FUNCTION_BLOCK Control (* Composite Function Block Type *)
  (* Standard: 61499-2 *)
  (* Version 0.0, 6/3/2016, Andrei, nxtControl GmbH, template *)
  PACKAGE Main;
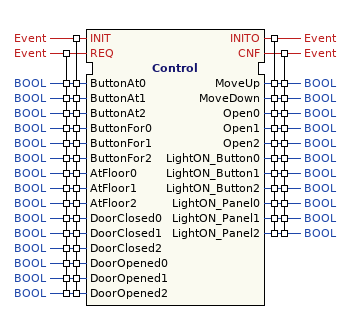
  EVENT_INPUT
    INIT WITH ButtonAt0, ButtonAt1, ButtonAt2, ButtonFor0, ButtonFor1, ButtonFor2, AtFloor0, AtFloor1, AtFloor2, DoorClosed0, DoorClosed1, DoorClosed2, DoorOpened0, DoorOpened1, DoorOpened2; (* Initialization Request *)
    REQ WITH ButtonAt0, ButtonAt1, ButtonAt2, ButtonFor0, ButtonFor1, ButtonFor2, AtFloor0, AtFloor1, AtFloor2, DoorClosed0, DoorClosed1, DoorClosed2, DoorOpened0, DoorOpened1, DoorOpened2; (* Normal Execution Request *)
  END_EVENT
  EVENT_OUTPUT
    INITO WITH MoveUp, MoveDown, Open0, Open1, Open2, LightON_Button0, LightON_Button1, LightON_Button2, LightON_Panel0, LightON_Panel1, LightON_Panel2; (* Initialization Confirm *)
    CNF WITH MoveUp, MoveDown, Open0, Open1, Open2, LightON_Button0, LightON_Button1, LightON_Button2, LightON_Panel0, LightON_Panel1, LightON_Panel2; (* Execution Confirmation *)
  END_EVENT
  VAR_INPUT
    ButtonAt0 : BOOL;
    ButtonAt1 : BOOL;
    ButtonAt2 : BOOL;
    ButtonFor0 : BOOL;
    ButtonFor1 : BOOL;
    ButtonFor2 : BOOL;
    AtFloor0 : BOOL; (* Input event qualifier *)
    AtFloor1 : BOOL;
    AtFloor2 : BOOL;
    DoorClosed0 : BOOL;
    DoorClosed1 : BOOL;
    DoorClosed2 : BOOL;
    DoorOpened0 : BOOL;
    DoorOpened1 : BOOL;
    DoorOpened2 : BOOL;
  END_VAR
  VAR_OUTPUT
    MoveUp : BOOL; (* Output event qualifier *)
    MoveDown : BOOL;
    Open0 : BOOL;
    Open1 : BOOL;
    Open2 : BOOL;
    LightON_Button0 : BOOL;
    LightON_Button1 : BOOL;
    LightON_Button2 : BOOL;
    LightON_Panel0 : BOOL;
    LightON_Panel1 : BOOL;
    LightON_Panel2 : BOOL;
  END_VAR
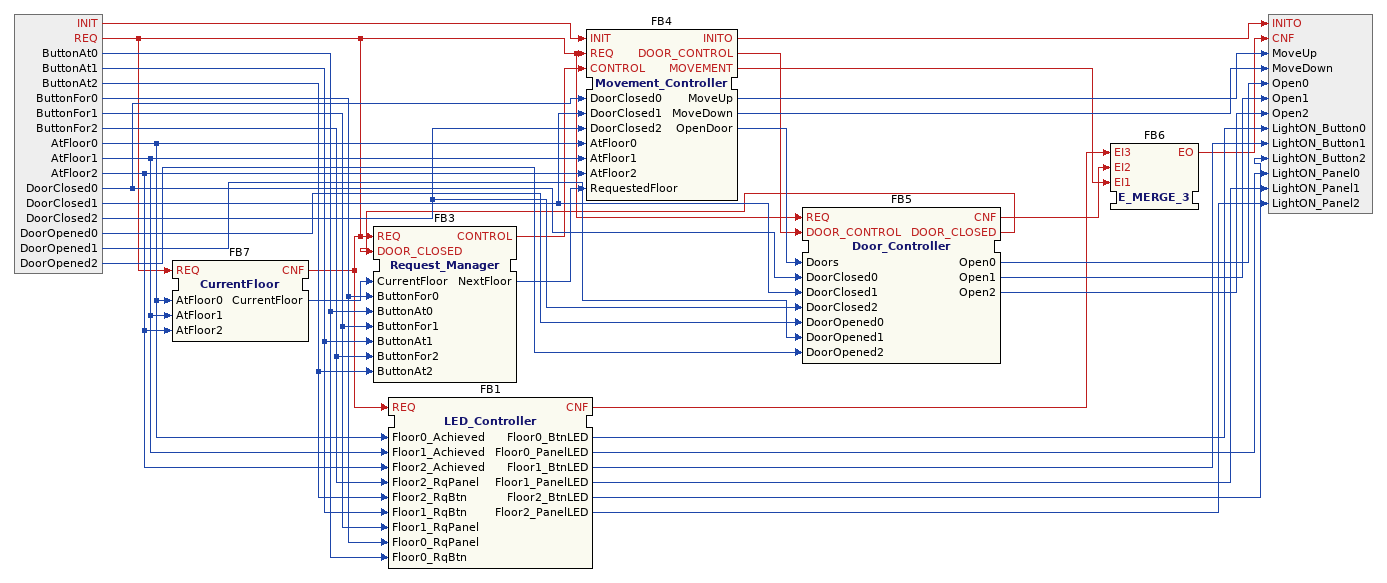
  FBS
    FB1 : LED_Controller;
    FB4 : Movement_Controller;
    FB5 : Door_Controller;
    FB6 : E_MERGE_3;
    FB3 : Request_Manager;
    FB7 : CurrentFloor;
  END_FBS
  EVENT_CONNECTIONS
    REQ TO FB1.REQ;
    FB4.INITO TO INITO;
    INIT TO FB4.INIT;
    REQ TO FB5.REQ;
    FB4.DOOR_CONTROL TO FB5.DOOR_CONTROL;
    FB1.CNF TO FB6.EI3;
    FB6.EO TO CNF;
    FB5.CNF TO FB6.EI2;
    FB4.MOVEMENT TO FB6.EI1;
    REQ TO FB4.REQ;
    FB3.CONTROL TO FB4.CONTROL;
    REQ TO FB7.REQ;
    REQ TO FB3.REQ;
    FB5.DOOR_CLOSED TO FB3.DOOR_CLOSED;
    FB7.CNF TO FB3.REQ;
  END_CONNECTIONS
  DATA_CONNECTIONS
    AtFloor0 TO FB1.Floor0_Achieved;
    AtFloor1 TO FB1.Floor1_Achieved;
    FB1.Floor0_BtnLED TO LightON_Button0;
    FB1.Floor0_PanelLED TO LightON_Panel0;
    FB1.Floor1_BtnLED TO LightON_Button1;
    FB1.Floor1_PanelLED TO LightON_Panel1;
    FB1.Floor2_BtnLED TO LightON_Button2;
    FB1.Floor2_PanelLED TO LightON_Panel2;
    AtFloor2 TO FB1.Floor2_Achieved;
    ButtonFor2 TO FB1.Floor2_RqPanel;
    ButtonAt2 TO FB1.Floor2_RqBtn;
    ButtonAt1 TO FB1.Floor1_RqBtn;
    ButtonFor1 TO FB1.Floor1_RqPanel;
    ButtonFor0 TO FB1.Floor0_RqPanel;
    ButtonAt0 TO FB1.Floor0_RqBtn;
    FB4.MoveUp TO MoveUp;
    FB4.MoveDown TO MoveDown;
    DoorClosed0 TO FB4.DoorClosed0;
    DoorClosed1 TO FB4.DoorClosed1;
    DoorClosed2 TO FB4.DoorClosed2;
    AtFloor0 TO FB4.AtFloor0;
    AtFloor1 TO FB4.AtFloor1;
    AtFloor2 TO FB4.AtFloor2;
    FB5.Open0 TO Open0;
    FB5.Open1 TO Open1;
    FB5.Open2 TO Open2;
    FB4.OpenDoor TO FB5.Doors;
    DoorClosed0 TO FB5.DoorClosed0;
    DoorClosed1 TO FB5.DoorClosed1;
    DoorClosed2 TO FB5.DoorClosed2;
    DoorOpened0 TO FB5.DoorOpened0;
    DoorOpened1 TO FB5.DoorOpened1;
    DoorOpened2 TO FB5.DoorOpened2;
    FB3.NextFloor TO FB4.RequestedFloor;
    AtFloor0 TO FB7.AtFloor0;
    AtFloor1 TO FB7.AtFloor1;
    AtFloor2 TO FB7.AtFloor2;
    FB7.CurrentFloor TO FB3.CurrentFloor;
    ButtonFor0 TO FB3.ButtonFor0;
    ButtonAt0 TO FB3.ButtonAt0;
    ButtonFor1 TO FB3.ButtonFor1;
    ButtonAt1 TO FB3.ButtonAt1;
    ButtonFor2 TO FB3.ButtonFor2;
    ButtonAt2 TO FB3.ButtonAt2;
  END_CONNECTIONS
END_FUNCTION_BLOCK
